// TIA Portal V18 export
FUNCTION "LED" : Void   // FC6, LAD
{ S7_Optimized_Access := 'TRUE' }
AUTHOR : HenriP
VERSION : 0.1
// stored: AutoNumber true, IsIECCheckEnabled false, SetENOAutomatically false, UDAEnableTagReadback false
   VAR_INPUT
      Green : Bool;
      GreenBlink : Bool;
      Red : Bool;
      RedBlink : Bool;
      RedGreen : Bool;
   END_VAR
   VAR_OUTPUT
      "Led Green" : Bool;
      "Led Red" : Bool;
   END_VAR
   VAR_TEMP
      RedGreenBlinkTemp : Bool;
      RedBlinkTemp : Bool;
      GreenBlinkTemp : Bool;
   END_VAR
BEGIN

REGION Network 1: Green Led
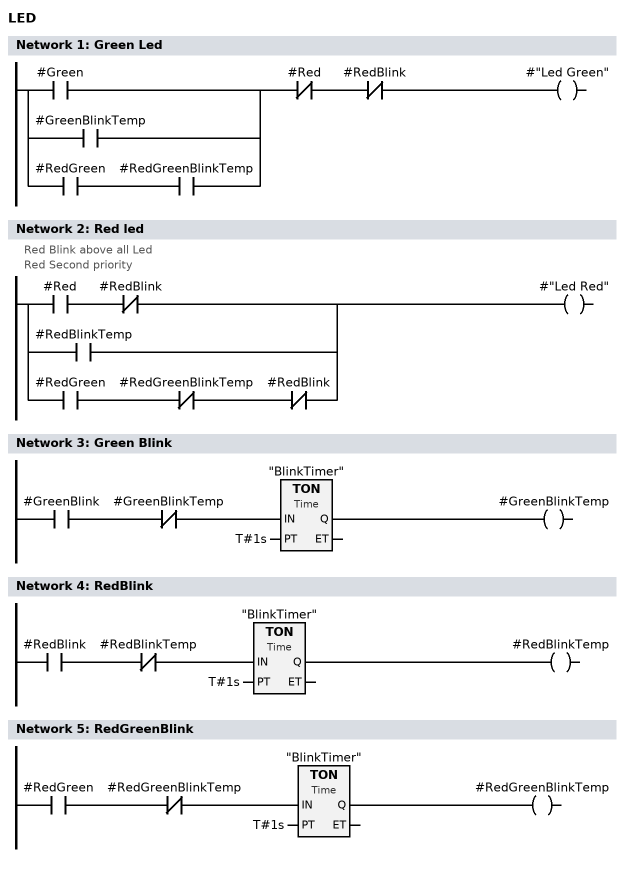
   RUNG wire#powerrail
      Contact( #Green )
      wire#w1
      I_Contact( #Red )
      I_Contact( #RedBlink )
      Coil( #"Led Green" )
   END_RUNG
   RUNG wire#powerrail
      Contact( #GreenBlinkTemp )
   END_RUNG wire#w1
   RUNG wire#powerrail
      Contact( #RedGreen )
      Contact( #RedGreenBlinkTemp )
   END_RUNG wire#w1
   // the same network as SCL:
   #"Led Green" := (#Green OR #GreenBlinkTemp OR (#RedGreen AND #RedGreenBlinkTemp)) AND NOT #Red AND NOT #RedBlink;
END_REGION

REGION Network 2: Red led
   // Red Blink above all Led
   // Red Second priority
   RUNG wire#powerrail
      Contact( #Red )
      I_Contact( #RedBlink )
      wire#w1
      Coil( #"Led Red" )
   END_RUNG
   RUNG wire#powerrail
      Contact( #RedBlinkTemp )
   END_RUNG wire#w1
   RUNG wire#powerrail
      Contact( #RedGreen )
      I_Contact( #RedGreenBlinkTemp )
      I_Contact( #RedBlink )
   END_RUNG wire#w1
   // the same network as SCL:
   #"Led Red" := (#Red AND NOT #RedBlink) OR #RedBlinkTemp OR (#RedGreen AND NOT #RedGreenBlinkTemp AND NOT #RedBlink);
END_REGION

REGION Network 3: Green Blink
   RUNG wire#powerrail
      Contact( #GreenBlink )
      I_Contact( #GreenBlinkTemp )
      { S7_Templates := "time_type := Time" } "BlinkTimer".TON(pt := T#1s, et =>)
      Coil( #GreenBlinkTemp )
   END_RUNG
   // the same network as SCL:
   "BlinkTimer".TON(IN := #GreenBlink AND NOT #GreenBlinkTemp, PT := T#1s);
   #GreenBlinkTemp := "BlinkTimer".Q;
END_REGION

REGION Network 4: RedBlink
   RUNG wire#powerrail
      Contact( #RedBlink )
      I_Contact( #RedBlinkTemp )
      { S7_Templates := "time_type := Time" } "BlinkTimer".TON(pt := T#1s, et =>)
      Coil( #RedBlinkTemp )
   END_RUNG
   // the same network as SCL:
   "BlinkTimer".TON(IN := #RedBlink AND NOT #RedBlinkTemp, PT := T#1s);
   #RedBlinkTemp := "BlinkTimer".Q;
END_REGION

REGION Network 5: RedGreenBlink
   RUNG wire#powerrail
      Contact( #RedGreen )
      I_Contact( #RedGreenBlinkTemp )
      { S7_Templates := "time_type := Time" } "BlinkTimer".TON(pt := T#1s, et =>)
      Coil( #RedGreenBlinkTemp )
   END_RUNG
   // the same network as SCL:
   "BlinkTimer".TON(IN := #RedGreen AND NOT #RedGreenBlinkTemp, PT := T#1s);
   #RedGreenBlinkTemp := "BlinkTimer".Q;
END_REGION
END_FUNCTION
